// SIMATIC STEP 7 (V5.x) project 2 IL Calc
// CPU: CPU 314C-2 PN/DP
// station: Hardware
// station: SIMATIC 300(1)
// station: P_ADR_BUS
// program: S7-Programm(1)

SYMBOL_TABLE
"HIGH IL1000"	I 2.0	BOOL
"LOW IL1000"	I 2.1	BOOL
"GO IL1000"	I 2.2	BOOL
"HH IL1000"	I 2.3	BOOL
"LL IL1000"	I 2.4	BOOL
"Messwert ungültig IL1000"	I 3.1	BOOL
"Messwert u Bereich 1000"	I 3.2	BOOL
"Messwert ü Bereich 1000"	I 3.3	BOOL
"Fehlerstatus IL1000"	I 3.7	BOOL
"Ext IN-Reaktion 1 IL1000"	I 4.0	BOOL
"Ext IN-Reaktion 2 IL1000"	I 4.1	BOOL
"Ext IN-Reaktion 3 IL1000"	I 4.2	BOOL
"Ext IN-Reaktion 4 IL1000"	I 4.3	BOOL
"HIGH IL1050"	I 9.0	BOOL
"LOW IL1050"	I 9.1	BOOL
"GO IL1050"	I 9.2	BOOL
"HH IL1050"	I 9.3	BOOL
"LL IL1050"	I 9.4	BOOL
"Messwert ungültig 1050"	I 10.1	BOOL
"Messwert u Bereich 1050"	I 10.2	BOOL
"Messwert ü Bereich 1050"	I 10.3	BOOL
"Fehlerstatus IL1050"	I 10.4	BOOL
"Ext IN-Reaktion 1 IL1050"	I 11.0	BOOL
"Ext IN-Reaktion 2 IL1050"	I 11.1	BOOL
"Ext IN-Reaktion 3 IL1050"	I 11.2	BOOL
"Ext IN-Reaktion 4 IL1050"	I 11.3	BOOL
"REQUEST SFB52"	I 136.0	BOOL
"REQUEST SFB53"	I 136.1	BOOL
"Messwert IL1000"	ID 5	DWORD
"Messwert IL1050"	ID 12	DWORD
"Done WRITE"	M 0.1	BOOL
"Busy WRITE"	M 0.2	BOOL
"Error WRITE"	M 0.3	BOOL
"Valid READ"	M 1.0	BOOL
"Busy READ"	M 1.1	BOOL
"Error READ"	M 1.2	BOOL
"Status WRITE"	MD 2	DWORD
"Status READ"	MD 6	DWORD
"Len"	MW 10	INT
"Ext IN Anf. 1 IL1000"	Q 1.0	BOOL
"Ext IN Anf. 2 IL1000"	Q 1.1	BOOL
"Ext IN Anf. 3 IL1000"	Q 1.2	BOOL
"Ext IN Anf. 4 IL1000"	Q 1.3	BOOL
"Ext IN Anf. 1 IL1050"	Q 2.0	BOOL
"Ext IN Anf. 2 IL1050"	Q 2.1	BOOL
"Ext IN Anf. 3 IL1050"	Q 2.2	BOOL
"Ext IN Anf. 4 IL1050"	Q 2.3	BOOL
"RDREC"	SFB 52	SFB 52	// Read a Process Data Record
"WRREC"	SFB 53	SFB 53	// Write a Process Data Record
"Variablentabelle_1"	VAT 1	
END_SYMBOL_TABLE

DATA_BLOCK DB 1
AUTHOR : SIMATIC
FAMILY : DP
VERSION : 0.1
"RDREC"
BEGIN
END_DATA_BLOCK

DATA_BLOCK DB 2
VERSION : 0.1
  STRUCT
   ReadRecord : ARRAY  [0 .. 20 ] OF //vorläufige Platzhaltervariable
   BYTE  := B#16#0;
  END_STRUCT ;	
BEGIN
END_DATA_BLOCK

DATA_BLOCK DB 3
AUTHOR : SIMATIC
FAMILY : DP
VERSION : 0.1
"WRREC"
BEGIN
END_DATA_BLOCK

DATA_BLOCK DB 4
VERSION : 0.1
  STRUCT
   WriteRecord : ARRAY  [0 .. 20 ] OF //vorläufige Platzhaltervariable
   DWORD  := DW#16#0;
  END_STRUCT ;	
BEGIN
END_DATA_BLOCK

ORGANIZATION_BLOCK OB 1
TITLE = "Main Program Sweep (Cycle)"
VERSION : 0.1
VAR_TEMP
  OB1_EV_CLASS : BYTE ;	//Bits 0-3 = 1 (Coming event), Bits 4-7 = 1 (Event class 1)
  OB1_SCAN_1 : BYTE ;	//1 (Cold restart scan 1 of OB 1), 3 (Scan 2-n of OB 1)
  OB1_PRIORITY : BYTE ;	//Priority of OB Execution
  OB1_OB_NUMBR : BYTE ;	//1 (Organization block 1, OB1)
  OB1_RESERVED_1 : BYTE ;	//Reserved for system
  OB1_RESERVED_2 : BYTE ;	//Reserved for system
  OB1_PREV_CYCLE : INT ;	//Cycle time of previous OB1 scan (milliseconds)
  OB1_MIN_CYCLE : INT ;	//Minimum cycle time of OB1 (milliseconds)
  OB1_MAX_CYCLE : INT ;	//Maximum cycle time of OB1 (milliseconds)
  OB1_DATE_TIME : DATE_AND_TIME ;	//Date and time OB1 started
END_VAR
BEGIN
NETWORK
TITLE =
      A     "REQUEST SFB52";
      =     L 20.0;
      BLD   103;
      BLD   9;
      =     L 25.0;
      CDB;
      OPN   DI 1;
      TAR2  LD 21;
      A     L 20.0;
      =     DIX 0.0;
      L     L#32769;
      T     DID 2;
      L     37;
      T     DIW 6;
      L     4;
      T     DIW 8;
      L     W#16#1002;
      T     DIW 18;
      L     4;
      T     DIW 20;
      L     2;
      T     DIW 22;
      L     P#DBX 0.0;
      T     DID 24;
      LAR2  P#DBX 0.0;
      UC    "RDREC";
      LAR2  LD 21;
      A     DIX 10.0;
      =     "Valid READ";
      A     DIX 10.1;
      =     "Busy READ";
      A     DIX 10.2;
      =     "Error READ";
      L     DID 12;
      T     "Status READ";
      L     DIW 16;
      T     "Len";
      CDB;
      BLD   10;
      NOP   0;
NETWORK
TITLE =
      A     "REQUEST SFB53";
      =     L 20.0;
      BLD   103;
      BLD   9;
      =     L 25.0;
      CDB;
      OPN   DI 3;
      TAR2  LD 21;
      A     L 20.0;
      =     DIX 0.0;
      L     L#32769;
      T     DID 2;
      L     1;
      T     DIW 6;
      L     4;
      T     DIW 8;
      L     W#16#1006;
      T     DIW 16;
      L     1;
      T     DIW 18;
      L     4;
      T     DIW 20;
      L     P#DBX 0.0;
      T     DID 22;
      LAR2  P#DBX 0.0;
      UC    "WRREC";
      LAR2  LD 21;
      A     DIX 10.0;
      =     "Done WRITE";
      A     DIX 10.1;
      =     "Busy WRITE";
      A     DIX 10.2;
      =     "Error WRITE";
      L     DID 12;
      T     "Status WRITE";
      CDB;
      BLD   10;
      NOP   0;
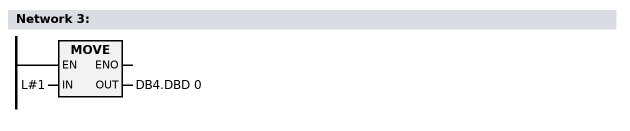
NETWORK
TITLE =
      L     L#1;
      T     DB4.DBD 0;
      NOP   0;
END_ORGANIZATION_BLOCK
